PROGRAM MAIN
VAR
	MoverMan	: FB_MoverMan;
END_VAR

_02_SAFETY();
_05_FLAGS( xIN_AIR:=TRUE, xIN_btRES_TEMP:=HMI.btArMain[8]);

//HMI
_10_HMI();

MoverMan();

//AUTO
_20_AUTO(xIN_Quit:= _14_STATE._FB_btQUIT.pbtIN^.rtrig , enIN_State:= HMI.enState);

//DJ Test
DEBUG();

END_PROGRAM

(* stored: Version 1.1.0.1, ProductVersion 3.1.4024.6
   POU MAIN: Id {dba9db14-aa7f-405f-8447-2b4bbb3b30dd}, SpecialFunc None *)
